// TIA Portal project "PLC Reload" (V17)

(* hardware
DEVICE "S7-1200 station_1"  S7-1200 Station
   slot 0: "Rack_0"  S7-1200 Rack  Rack  V1.0
   slot 1: "PLC_1"  CPU 1215C DC/DC/Rly  6ES7 215-1HG40-0XB0  V4.2
   slot 2: "DI 16x24VDC/DQ 16xRelay_1"  SM 1223 DI16/DQ16 x relay  6ES7 223-1PL32-0XB0  V2.0
   slot 3: "AI 4x13BIT_1"  6ES7 231-4HD32-0XB0  V2.1
*)

// ===== PLC "PLC_1"  CPU 1215C DC/DC/Rly =====

VAR_GLOBAL   // PLC tag table "Default tag table"
   "bt.Auto" AT %I0.1 : Bool;
   "CTHT_Thuan" AT %I1.2 : Bool;
   "bt.Manual" AT %I0.2 : Bool;
   "Sensor 1 Nhiệt Độ" AT %IW64 : Int;
   "Sensor 1 Độ Ảm" AT %IW66 : Int;
   "Tag_15" AT %IW11 : Int;
   "Sensor 2 Nhiệt Độ" AT %IW112 : Int;
   "Sensor 2 Độ Ảm" AT %IW114 : Int;
   "Sensor 3 Nhiệt Độ" AT %IW116 : Int;
   "Sensor 3 Độ Ảm" AT %IW118 : Int;
   "bt.BangTai" AT %I0.3 : Bool;
   "bt.Manual Đèn 1 3" AT %I0.5 : Bool;
   "bt. Cylanh Thức Ăn" AT %I0.4 : Bool;
   "CTHT_Nguoc" AT %I1.1 : Bool;
   "bt.Manual Đèn 2 4" AT %I0.6 : Bool;
   "bt.Quat" AT %I0.7 : Bool;
   "bt.PhunSuong" AT %I1.0 : Bool;
   "Đèn sưởi 1" AT %Q1.0 : Bool;
   "Băng tải 1" AT %Q1.1 : Bool;
   "#R Pump" AT %Q8.0 : Bool;
   "Xy Lanh An Duoi" AT %Q0.5 : Bool;
   "QuatAm2" AT %Q0.6 : Bool;
   "QuatAm1" AT %Q8.1 : Bool;
   "Van trên 2" AT %Q8.2 : Bool;
   "QuatThoi_Duoi" AT %Q9.1 : Bool;
   "QuatHutAm_Duoi" AT %Q9.2 : Bool;
   "Đèn sưởi 2" AT %Q0.7 : Bool;
   "#R Motor Fwd" AT %Q0.3 : Bool;
   "#R Motor Rev" AT %Q0.4 : Bool;
   "Light Green" AT %Q0.0 : Bool;
   "Light Yellow" AT %Q0.2 : Bool;
   "Băng tải 3" AT %Q9.3 : Bool;
   "Băng tải 4" AT %Q9.4 : Bool;
   "Băng tải 2" AT %Q9.0 : Bool;
   "Xylanh an tren" AT %Q8.6 : Bool;
   "Xylanh Nâng" AT %Q8.7 : Bool;
   "Tag_33" AT %Q2.4 : Bool;
   "Tag_35" AT %Q2.5 : Bool;
   "Van 3 - Bồn" AT %Q8.3 : Bool;
   "Van trên 4" AT %Q8.4 : Bool;
   "Van 1,5" AT %Q8.5 : Bool;
   "System_Byte" AT %MB100 : Byte;
   "FirstScan" AT %M100.0 : Bool;
   "DiagStatusUpdate" AT %M100.1 : Bool;
   "AlwaysTRUE" AT %M100.2 : Bool;
   "AlwaysFALSE" AT %M100.3 : Bool;
   "Clock_Byte" AT %MB110 : Byte;
   "Clock_10Hz" AT %M110.0 : Bool;
   "Clock_5Hz" AT %M110.1 : Bool;
   "Clock_2.5Hz" AT %M110.2 : Bool;
   "Clock_2Hz" AT %M110.3 : Bool;
   "Clock_1.25Hz" AT %M110.4 : Bool;
   "Clock_1Hz" AT %M110.5 : Bool;
   "Clock_0.625Hz" AT %M110.6 : Bool;
   "Clock_0.5Hz" AT %M110.7 : Bool;
   "R #01 Test" AT %M0.0 : Bool;
   "m0.7" AT %M0.1 : Bool;
   "Tag_2" AT %M10.0 : Bool;
   "Tag_6" AT %M10.1 : Bool;
   "Tag_5" AT %M10.2 : Bool;
   "Tag_8" AT %M10.3 : Bool;
   "Tag_12" AT %M10.4 : Bool;
   "Tag_13" AT %M10.5 : Bool;
   "Tag_14" AT %M10.6 : Bool;
   "Tag_16" AT %M10.7 : Bool;
   "Tag_18" AT %M11.0 : Bool;
   "R #02 Test" AT %M11.1 : Bool;
   "ND NORM_1" AT %MD200 : Real;
   "DATA NhietDo_1" AT %MD204 : Real;
   "DA NORM 1" AT %MD208 : Real;
   "DATA DoAm_1" AT %MD212 : Real;
   "Tag_22" AT %MD216 : Real;
   "ND NORM_2" AT %MD220 : Real;
   "DATA NhietDo_2" AT %MD224 : Real;
   "DA NORM 2" AT %MD228 : Real;
   "DATA DoAm_2" AT %MD232 : Real;
   "ND NORM_3" AT %MD440 : Real;
   "DATA NhietDo_3" AT %MD444 : Real;
   "DA NORM 3" AT %MD448 : Real;
   "DATA DoAm_3" AT %MD452 : Real;
   "Auto Mode" AT %M1.0 : Bool;
   "Manual Mode" AT %M1.1 : Bool;
   "Cylanh Nâng" AT %M2.0 : Bool;
   "Manual Băng Tải" AT %M1.2 : Bool;
   "Băng Tải 1 2 Run" AT %M2.1 : Bool;
   "Tag_4" AT %M0.7 : Bool;
   "Tag_19" AT %M0.6 : Bool;
   "Manual Cylanh Thức Ăn" AT %M1.3 : Bool;
   "Cylanh Up Thuc Ăn" AT %M2.2 : Bool;
   "Motor FWD" AT %M2.4 : Bool;
   "Motor REV" AT %M2.5 : Bool;
   "Tag_36" AT %M6.0 : Bool;
   "Tag_37" AT %M2.3 : Bool;
   "Đèn 1 3 Manual" AT %M1.4 : Bool;
   "Đèn 2 4 Manual" AT %M1.5 : Bool;
   "Manual Quạt" AT %M1.6 : Bool;
   "Manual Phun Sương" AT %M1.7 : Bool;
   "Pump Run" AT %M2.6 : Bool;
   "Van chuong 1" AT %M2.7 : Bool;
   "Van chuong 2" AT %M3.0 : Bool;
   "Van chuong 3,4" AT %M3.1 : Bool;
   "Van 4" AT %M3.2 : Bool;
   "Van lên bồn" AT %M3.3 : Bool;
   "Auto Buổi Sáng" AT %M4.0 : Bool;
   "Auto Buổi Trưa" AT %M4.1 : Bool;
   "Auto Buổi Chiều" AT %M4.2 : Bool;
   "Auto Theo Buổi" AT %M5.0 : Bool;
   "TG_Nhiet_1" AT %M5.1 : Bool;
   "Mode Theo Buổi" AT %M5.2 : Bool;
   "Mode Cảm Biến + Theo Buổi" AT %M5.3 : Bool;
   "Tag_7" AT %MD304 : Real;
   "Tag_9" AT %MD312 : Real;
   "Tag_10" AT %MD324 : Real;
   "Tag_11" AT %MD332 : Real;
   "Tag_20" AT %MD344 : Real;
   "Tag_21" AT %MD352 : Real;
   "TG_Nhiet_2" AT %M5.4 : Bool;
   "TG_Nhiet_3" AT %M5.5 : Bool;
   "Mode Cảm Biến + Theo Buổi R" AT %M5.6 : Bool;
   "Tag_1" AT %M88.4 : Bool;
   "Tag_23" AT %M778.6 : Bool;
   "Cho an Tren" AT %M12.0 : Bool;
   "Don Ve Sinh" AT %M12.1 : Bool;
   "TG_Am_1" AT %M7.0 : Bool;
   "Tag_25" AT %MD404 : Real;
   "Tag_26" AT %MD412 : Real;
   "Tag_27" AT %MD424 : Real;
   "Tag_28" AT %MD432 : Real;
   "TG_Am_2" AT %M7.1 : Bool;
   "TG_Am_3" AT %M7.2 : Bool;
   "Tag_24" AT %M864.4 : Bool;
   "Tag_29" AT %M54.7 : Bool;
   "Sensor Pump Done" AT %I1.3 : Bool;
   "TG_Am_Quat_1" AT %M7.5 : Bool;
   "TG_Am_Quat_3" AT %M7.6 : Bool;
   "TG_Am_Quat_2" AT %M7.7 : Bool;
   "Tag_17" AT %M8.1 : Bool;
   "DonVSTren" AT %M12.2 : Bool;
END_VAR

DATA_BLOCK "Time"   // DB6
{ S7_Optimized_Access := 'TRUE' }
VERSION : 0.1
   VAR
      Reatime : DTL;
      "Dọn Vệ Sinh Trên 1" : Bool;
      Retval : Int;
      "Ăn Dưới 1" : Bool;
      "An 2" : Bool;
      "An 3" : Bool;
      "Ăn Trên 1" : Bool;
      "An Tren 2" : Bool;
      "An Tren 3" : Bool;
      "An Tren 4" : Bool;
      "An Tren 5" : Bool;
      "Dọn Vệ Sinh Dưới 1" : Bool;
      "Don VS Duoi 2" : Bool;
   END_VAR
BEGIN
END_DATA_BLOCK

DATA_BLOCK "Temp"   // DB13
{ S7_Optimized_Access := 'FALSE' }
VERSION : 0.1
   VAR
      DataNhiet1 : Real;
      DataNhiet2 : Real;
      DataNhiet3 : Real;
      DataAm1 : Real;
      DataAm2 : Real;
      DataAm3 : Real;
      SetNhiet1 : Real;
      SetNhiet2 : Real;
      SetNhiet3 : Real;
      SetAm1 : Real;
      SetAm2 : Real;
      SetAm3 : Real;
   END_VAR
BEGIN
END_DATA_BLOCK

// folder: System blocks/Program resources

DATA_BLOCK "Delay Thưc Ăn"   // DB1
{ S7_Optimized_Access := 'TRUE' }
AUTHOR : Simatic
FAMILY : IEC
NAME : IEC_TMR
VERSION : 1.0
// stored: InstanceOfName IEC_TIMER
"IEC_TIMER"
BEGIN
END_DATA_BLOCK

DATA_BLOCK "Cylanh Nâng DL"   // DB2
{ S7_Optimized_Access := 'TRUE' }
AUTHOR : Simatic
FAMILY : IEC
NAME : IEC_TMR
VERSION : 1.0
// stored: InstanceOfName IEC_TIMER
"IEC_TIMER"
BEGIN
END_DATA_BLOCK

DATA_BLOCK "Motor Check FWD"   // DB3
{ S7_Optimized_Access := 'TRUE' }
AUTHOR : Simatic
FAMILY : IEC
NAME : IEC_TMR
VERSION : 1.0
// stored: InstanceOfName IEC_TIMER
"IEC_TIMER"
BEGIN
END_DATA_BLOCK

DATA_BLOCK "Motor Check REV"   // DB4
{ S7_Optimized_Access := 'TRUE' }
AUTHOR : Simatic
FAMILY : IEC
NAME : IEC_TMR
VERSION : 1.0
// stored: InstanceOfName IEC_TIMER
"IEC_TIMER"
BEGIN
END_DATA_BLOCK

DATA_BLOCK "Delay Pump"   // DB5
{ S7_Optimized_Access := 'TRUE' }
AUTHOR : Simatic
FAMILY : IEC
NAME : IEC_TMR
VERSION : 1.0
// stored: InstanceOfName IEC_TIMER
"IEC_TIMER"
BEGIN
END_DATA_BLOCK

DATA_BLOCK "Dl Time"   // DB7
{ S7_Optimized_Access := 'TRUE' }
AUTHOR : Simatic
FAMILY : IEC
NAME : IEC_TMR
VERSION : 1.0
// stored: InstanceOfName IEC_TIMER
"IEC_TIMER"
BEGIN
END_DATA_BLOCK

DATA_BLOCK "Dl Don Ve Sinh"   // DB8
{ S7_Optimized_Access := 'TRUE' }
AUTHOR : Simatic
FAMILY : IEC
NAME : IEC_TMR
VERSION : 1.0
// stored: InstanceOfName IEC_TIMER
"IEC_TIMER"
BEGIN
END_DATA_BLOCK

DATA_BLOCK "Dl Off"   // DB9
{ S7_Optimized_Access := 'TRUE' }
AUTHOR : Simatic
FAMILY : IEC
NAME : IEC_TMR
VERSION : 1.0
// stored: InstanceOfName IEC_TIMER
"IEC_TIMER"
BEGIN
END_DATA_BLOCK

DATA_BLOCK "DL Off 2"   // DB10
{ S7_Optimized_Access := 'TRUE' }
AUTHOR : Simatic
FAMILY : IEC
NAME : IEC_TMR
VERSION : 1.0
// stored: InstanceOfName IEC_TIMER
"IEC_TIMER"
BEGIN
END_DATA_BLOCK

DATA_BLOCK "DLOff 3"   // DB11
{ S7_Optimized_Access := 'TRUE' }
AUTHOR : Simatic
FAMILY : IEC
NAME : IEC_TMR
VERSION : 1.0
// stored: InstanceOfName IEC_TIMER
"IEC_TIMER"
BEGIN
END_DATA_BLOCK

DATA_BLOCK "DL Off Time An"   // DB12
{ S7_Optimized_Access := 'TRUE' }
AUTHOR : Simatic
FAMILY : IEC
NAME : IEC_TMR
VERSION : 1.0
// stored: InstanceOfName IEC_TIMER
"IEC_TIMER"
BEGIN
END_DATA_BLOCK

DATA_BLOCK "VESINH"   // DB14
{ S7_Optimized_Access := 'TRUE' }
AUTHOR : Simatic
FAMILY : IEC
NAME : IEC_TMR
VERSION : 1.0
// stored: InstanceOfName IEC_TIMER
"IEC_TIMER"
BEGIN
END_DATA_BLOCK

// folder: (top level)

FUNCTION "MC_Output" : Void   // FC1, LAD
{ S7_Optimized_Access := 'TRUE' }
VERSION : 0.1
BEGIN

REGION Network 1
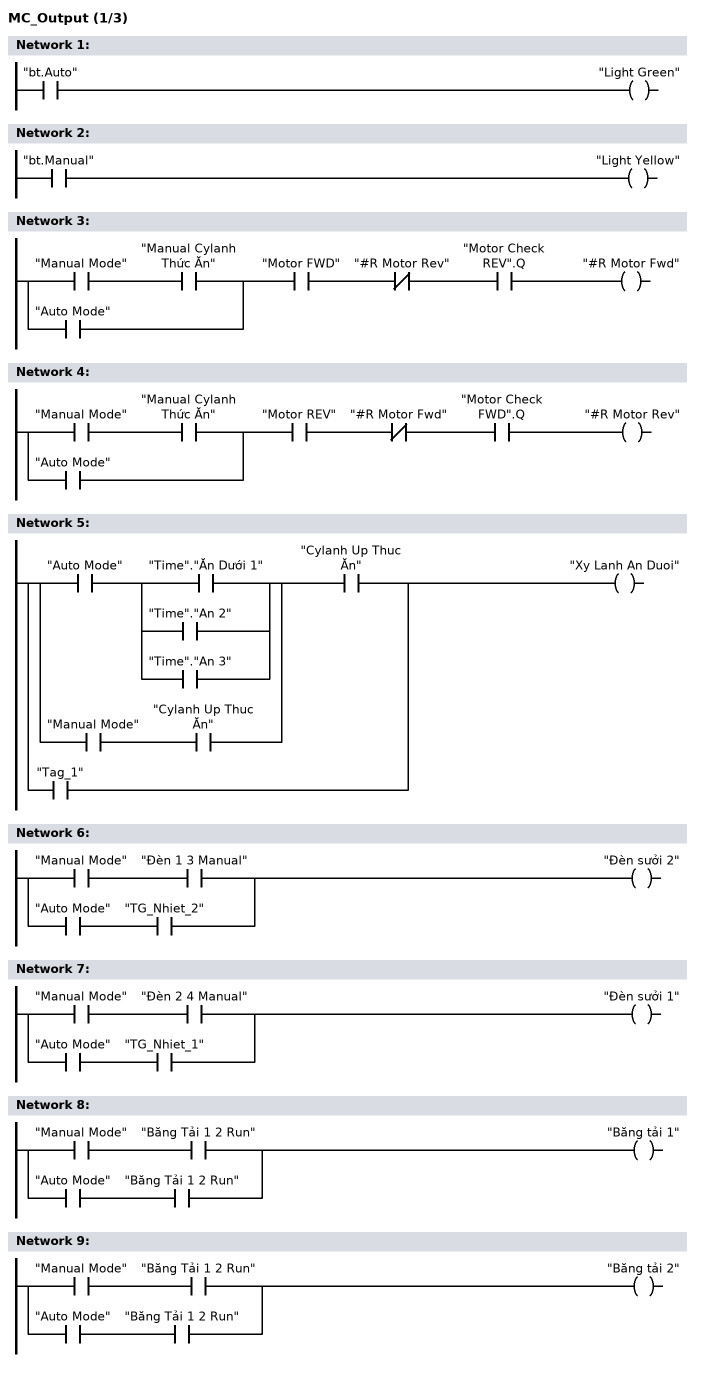
   RUNG wire#powerrail
      Contact( "bt.Auto" )
      Coil( "Light Green" )
   END_RUNG
   // the same network as SCL:
   "Light Green" := "bt.Auto";
END_REGION

REGION Network 2
   RUNG wire#powerrail
      Contact( "bt.Manual" )
      Coil( "Light Yellow" )
   END_RUNG
   // the same network as SCL:
   "Light Yellow" := "bt.Manual";
END_REGION

REGION Network 3
   RUNG wire#powerrail
      Contact( "Manual Mode" )
      Contact( "Manual Cylanh Thức Ăn" )
      wire#w1
      Contact( "Motor FWD" )
      I_Contact( "#R Motor Rev" )
      Contact( "Motor Check REV".Q )
      Coil( "#R Motor Fwd" )
   END_RUNG
   RUNG wire#powerrail
      Contact( "Auto Mode" )
   END_RUNG wire#w1
   // the same network as SCL:
   "#R Motor Fwd" := (("Manual Mode" AND "Manual Cylanh Thức Ăn") OR "Auto Mode") AND "Motor FWD" AND NOT "#R Motor Rev" AND "Motor Check REV".Q;
END_REGION

REGION Network 4
   RUNG wire#powerrail
      Contact( "Manual Mode" )
      Contact( "Manual Cylanh Thức Ăn" )
      wire#w1
      Contact( "Motor REV" )
      I_Contact( "#R Motor Fwd" )
      Contact( "Motor Check FWD".Q )
      Coil( "#R Motor Rev" )
   END_RUNG
   RUNG wire#powerrail
      Contact( "Auto Mode" )
   END_RUNG wire#w1
   // the same network as SCL:
   "#R Motor Rev" := (("Manual Mode" AND "Manual Cylanh Thức Ăn") OR "Auto Mode") AND "Motor REV" AND NOT "#R Motor Fwd" AND "Motor Check FWD".Q;
END_REGION

REGION Network 5
   RUNG wire#powerrail
      Contact( "Auto Mode" )
      wire#w1
      Contact( "Time"."Ăn Dưới 1" )
      wire#w2
      Contact( "Cylanh Up Thuc Ăn" )
      wire#w3
      Coil( "Xy Lanh An Duoi" )
   END_RUNG
   RUNG wire#w1
      Contact( "Time"."An 2" )
   END_RUNG wire#w2
   RUNG wire#w1
      Contact( "Time"."An 3" )
   END_RUNG wire#w2
   RUNG wire#powerrail
      Contact( "Manual Mode" )
      Contact( "Cylanh Up Thuc Ăn" )
   END_RUNG wire#w2
   RUNG wire#powerrail
      Contact( "Tag_1" )
   END_RUNG wire#w3
   // the same network as SCL:
   "Xy Lanh An Duoi" := ((("Auto Mode" AND ("Time"."Ăn Dưới 1" OR "Time"."An 2" OR "Time"."An 3")) OR ("Manual Mode" AND "Cylanh Up Thuc Ăn")) AND "Cylanh Up Thuc Ăn") OR "Tag_1";
END_REGION

REGION Network 6
   RUNG wire#powerrail
      Contact( "Manual Mode" )
      Contact( "Đèn 1 3 Manual" )
      wire#w1
      Coil( "Đèn sưởi 2" )
   END_RUNG
   RUNG wire#powerrail
      Contact( "Auto Mode" )
      Contact( "TG_Nhiet_2" )
   END_RUNG wire#w1
   // the same network as SCL:
   "Đèn sưởi 2" := ("Manual Mode" AND "Đèn 1 3 Manual") OR ("Auto Mode" AND "TG_Nhiet_2");
END_REGION

REGION Network 7
   RUNG wire#powerrail
      Contact( "Manual Mode" )
      Contact( "Đèn 2 4 Manual" )
      wire#w1
      Coil( "Đèn sưởi 1" )
   END_RUNG
   RUNG wire#powerrail
      Contact( "Auto Mode" )
      Contact( "TG_Nhiet_1" )
   END_RUNG wire#w1
   // the same network as SCL:
   "Đèn sưởi 1" := ("Manual Mode" AND "Đèn 2 4 Manual") OR ("Auto Mode" AND "TG_Nhiet_1");
END_REGION

REGION Network 8
   RUNG wire#powerrail
      Contact( "Manual Mode" )
      Contact( "Băng Tải 1 2 Run" )
      wire#w1
      Coil( "Băng tải 1" )
   END_RUNG
   RUNG wire#powerrail
      Contact( "Auto Mode" )
      Contact( "Băng Tải 1 2 Run" )
   END_RUNG wire#w1
   // the same network as SCL:
   "Băng tải 1" := ("Manual Mode" AND "Băng Tải 1 2 Run") OR ("Auto Mode" AND "Băng Tải 1 2 Run");
END_REGION

REGION Network 9
   RUNG wire#powerrail
      Contact( "Manual Mode" )
      Contact( "Băng Tải 1 2 Run" )
      wire#w1
      Coil( "Băng tải 2" )
   END_RUNG
   RUNG wire#powerrail
      Contact( "Auto Mode" )
      Contact( "Băng Tải 1 2 Run" )
   END_RUNG wire#w1
   // the same network as SCL:
   "Băng tải 2" := ("Manual Mode" AND "Băng Tải 1 2 Run") OR ("Auto Mode" AND "Băng Tải 1 2 Run");
END_REGION

REGION Network 10
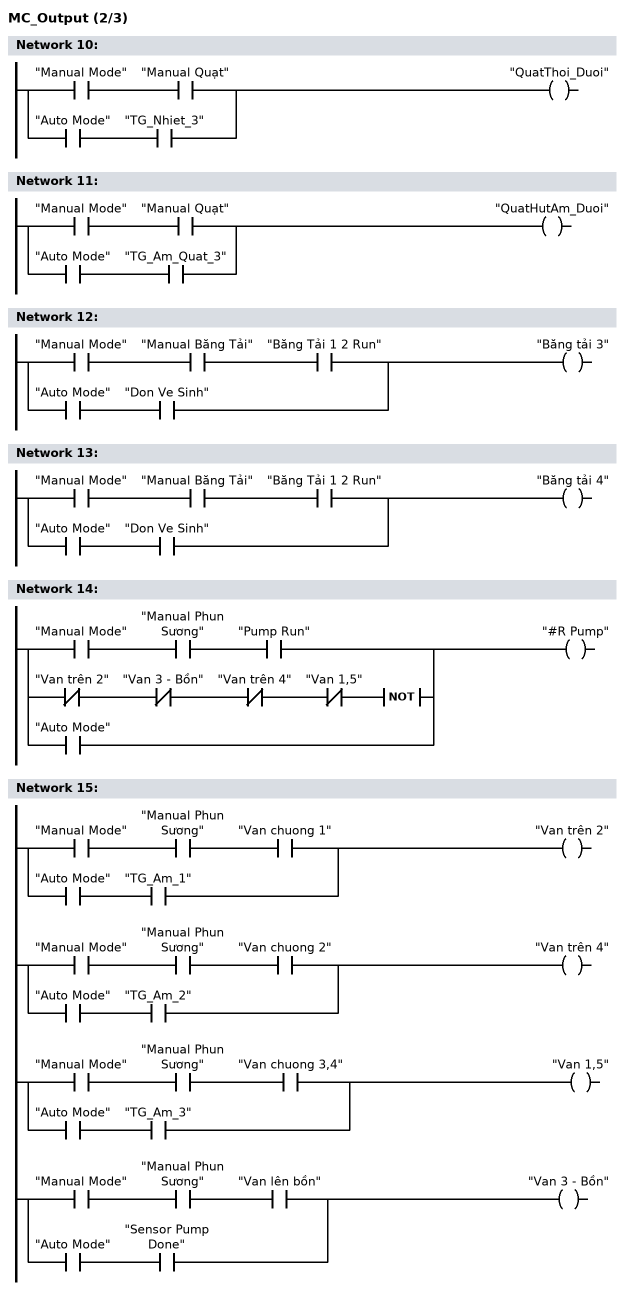
   RUNG wire#powerrail
      Contact( "Manual Mode" )
      Contact( "Manual Quạt" )
      wire#w1
      Coil( "QuatThoi_Duoi" )
   END_RUNG
   RUNG wire#powerrail
      Contact( "Auto Mode" )
      Contact( "TG_Nhiet_3" )
   END_RUNG wire#w1
   // the same network as SCL:
   "QuatThoi_Duoi" := ("Manual Mode" AND "Manual Quạt") OR ("Auto Mode" AND "TG_Nhiet_3");
END_REGION

REGION Network 11
   RUNG wire#powerrail
      Contact( "Manual Mode" )
      Contact( "Manual Quạt" )
      wire#w1
      Coil( "QuatHutAm_Duoi" )
   END_RUNG
   RUNG wire#powerrail
      Contact( "Auto Mode" )
      Contact( "TG_Am_Quat_3" )
   END_RUNG wire#w1
   // the same network as SCL:
   "QuatHutAm_Duoi" := ("Manual Mode" AND "Manual Quạt") OR ("Auto Mode" AND "TG_Am_Quat_3");
END_REGION

REGION Network 12
   RUNG wire#powerrail
      Contact( "Manual Mode" )
      Contact( "Manual Băng Tải" )
      Contact( "Băng Tải 1 2 Run" )
      wire#w1
      Coil( "Băng tải 3" )
   END_RUNG
   RUNG wire#powerrail
      Contact( "Auto Mode" )
      Contact( "Don Ve Sinh" )
   END_RUNG wire#w1
   // the same network as SCL:
   "Băng tải 3" := ("Manual Mode" AND "Manual Băng Tải" AND "Băng Tải 1 2 Run") OR ("Auto Mode" AND "Don Ve Sinh");
END_REGION

REGION Network 13
   RUNG wire#powerrail
      Contact( "Manual Mode" )
      Contact( "Manual Băng Tải" )
      Contact( "Băng Tải 1 2 Run" )
      wire#w1
      Coil( "Băng tải 4" )
   END_RUNG
   RUNG wire#powerrail
      Contact( "Auto Mode" )
      Contact( "Don Ve Sinh" )
   END_RUNG wire#w1
   // the same network as SCL:
   "Băng tải 4" := ("Manual Mode" AND "Manual Băng Tải" AND "Băng Tải 1 2 Run") OR ("Auto Mode" AND "Don Ve Sinh");
END_REGION

REGION Network 14
   RUNG wire#powerrail
      Contact( "Manual Mode" )
      Contact( "Manual Phun Sương" )
      Contact( "Pump Run" )
      wire#w1
      Coil( "#R Pump" )
   END_RUNG
   RUNG wire#powerrail
      I_Contact( "Van trên 2" )
      I_Contact( "Van 3 - Bồn" )
      I_Contact( "Van trên 4" )
      I_Contact( "Van 1,5" )
      Not()
   END_RUNG wire#w1
   RUNG wire#powerrail
      Contact( "Auto Mode" )
   END_RUNG wire#w1
   // the same network as SCL:
   "#R Pump" := ("Manual Mode" AND "Manual Phun Sương" AND "Pump Run") OR NOT (NOT "Van trên 2" AND NOT "Van 3 - Bồn" AND NOT "Van trên 4" AND NOT "Van 1,5") OR "Auto Mode";
END_REGION

REGION Network 15
   RUNG wire#powerrail
      Contact( "Manual Mode" )
      Contact( "Manual Phun Sương" )
      Contact( "Van chuong 1" )
      wire#w1
      Coil( "Van trên 2" )
   END_RUNG
   RUNG wire#powerrail
      Contact( "Auto Mode" )
      Contact( "TG_Am_1" )
   END_RUNG wire#w1
   RUNG wire#powerrail
      Contact( "Manual Mode" )
      Contact( "Manual Phun Sương" )
      Contact( "Van chuong 2" )
      wire#w2
      Coil( "Van trên 4" )
   END_RUNG
   RUNG wire#powerrail
      Contact( "Auto Mode" )
      Contact( "TG_Am_2" )
   END_RUNG wire#w2
   RUNG wire#powerrail
      Contact( "Manual Mode" )
      Contact( "Manual Phun Sương" )
      Contact( "Van chuong 3,4" )
      wire#w3
      Coil( "Van 1,5" )
   END_RUNG
   RUNG wire#powerrail
      Contact( "Auto Mode" )
      Contact( "TG_Am_3" )
   END_RUNG wire#w3
   RUNG wire#powerrail
      Contact( "Manual Mode" )
      Contact( "Manual Phun Sương" )
      Contact( "Van lên bồn" )
      wire#w4
      Coil( "Van 3 - Bồn" )
   END_RUNG
   RUNG wire#powerrail
      Contact( "Auto Mode" )
      Contact( "Sensor Pump Done" )
   END_RUNG wire#w4
   // the same network as SCL:
   "Van trên 2" := ("Manual Mode" AND "Manual Phun Sương" AND "Van chuong 1") OR ("Auto Mode" AND "TG_Am_1");
   "Van trên 4" := ("Manual Mode" AND "Manual Phun Sương" AND "Van chuong 2") OR ("Auto Mode" AND "TG_Am_2");
   "Van 1,5" := ("Manual Mode" AND "Manual Phun Sương" AND "Van chuong 3,4") OR ("Auto Mode" AND "TG_Am_3");
   "Van 3 - Bồn" := ("Manual Mode" AND "Manual Phun Sương" AND "Van lên bồn") OR ("Auto Mode" AND "Sensor Pump Done");
END_REGION

REGION Network 17
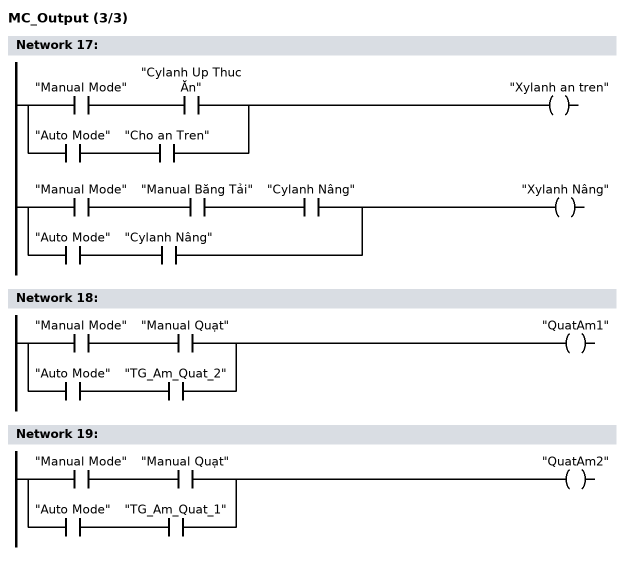
   RUNG wire#powerrail
      Contact( "Manual Mode" )
      Contact( "Cylanh Up Thuc Ăn" )
      wire#w1
      Coil( "Xylanh an tren" )
   END_RUNG
   RUNG wire#powerrail
      Contact( "Auto Mode" )
      Contact( "Cho an Tren" )
   END_RUNG wire#w1
   RUNG wire#powerrail
      Contact( "Manual Mode" )
      Contact( "Manual Băng Tải" )
      Contact( "Cylanh Nâng" )
      wire#w2
      Coil( "Xylanh Nâng" )
   END_RUNG
   RUNG wire#powerrail
      Contact( "Auto Mode" )
      Contact( "Cylanh Nâng" )
   END_RUNG wire#w2
   // the same network as SCL:
   "Xylanh an tren" := ("Manual Mode" AND "Cylanh Up Thuc Ăn") OR ("Auto Mode" AND "Cho an Tren");
   "Xylanh Nâng" := ("Manual Mode" AND "Manual Băng Tải" AND "Cylanh Nâng") OR ("Auto Mode" AND "Cylanh Nâng");
END_REGION

REGION Network 18
   RUNG wire#powerrail
      Contact( "Manual Mode" )
      Contact( "Manual Quạt" )
      wire#w1
      Coil( "QuatAm1" )
   END_RUNG
   RUNG wire#powerrail
      Contact( "Auto Mode" )
      Contact( "TG_Am_Quat_2" )
   END_RUNG wire#w1
   // the same network as SCL:
   "QuatAm1" := ("Manual Mode" AND "Manual Quạt") OR ("Auto Mode" AND "TG_Am_Quat_2");
END_REGION

REGION Network 19
   RUNG wire#powerrail
      Contact( "Manual Mode" )
      Contact( "Manual Quạt" )
      wire#w1
      Coil( "QuatAm2" )
   END_RUNG
   RUNG wire#powerrail
      Contact( "Auto Mode" )
      Contact( "TG_Am_Quat_1" )
   END_RUNG wire#w1
   // the same network as SCL:
   "QuatAm2" := ("Manual Mode" AND "Manual Quạt") OR ("Auto Mode" AND "TG_Am_Quat_1");
END_REGION
END_FUNCTION

FUNCTION "MC_Input" : Void   // FC2, LAD
{ S7_Optimized_Access := 'TRUE' }
VERSION : 0.1
BEGIN

REGION Network 1
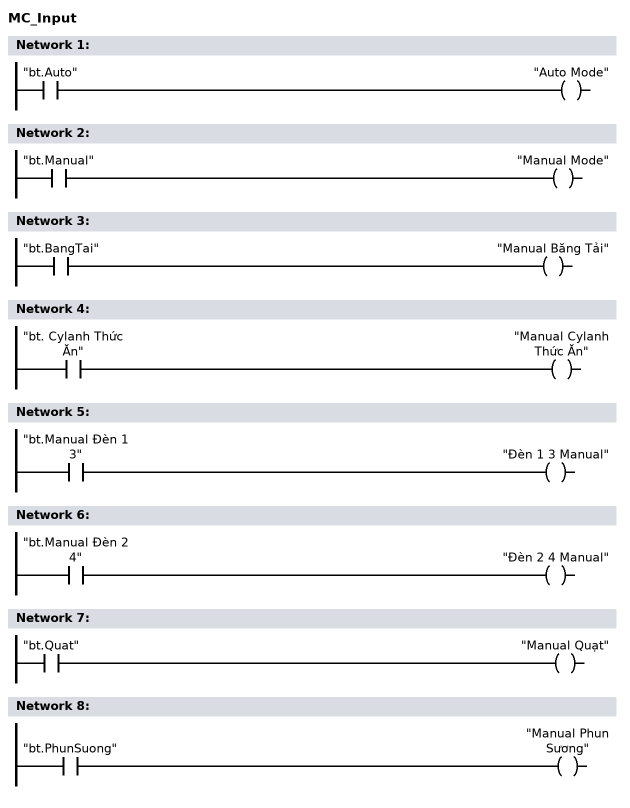
   RUNG wire#powerrail
      Contact( "bt.Auto" )
      Coil( "Auto Mode" )
   END_RUNG
   // the same network as SCL:
   "Auto Mode" := "bt.Auto";
END_REGION

REGION Network 2
   RUNG wire#powerrail
      Contact( "bt.Manual" )
      Coil( "Manual Mode" )
   END_RUNG
   // the same network as SCL:
   "Manual Mode" := "bt.Manual";
END_REGION

REGION Network 3
   RUNG wire#powerrail
      Contact( "bt.BangTai" )
      Coil( "Manual Băng Tải" )
   END_RUNG
   // the same network as SCL:
   "Manual Băng Tải" := "bt.BangTai";
END_REGION

REGION Network 4
   RUNG wire#powerrail
      Contact( "bt. Cylanh Thức Ăn" )
      Coil( "Manual Cylanh Thức Ăn" )
   END_RUNG
   // the same network as SCL:
   "Manual Cylanh Thức Ăn" := "bt. Cylanh Thức Ăn";
END_REGION

REGION Network 5
   RUNG wire#powerrail
      Contact( "bt.Manual Đèn 1 3" )
      Coil( "Đèn 1 3 Manual" )
   END_RUNG
   // the same network as SCL:
   "Đèn 1 3 Manual" := "bt.Manual Đèn 1 3";
END_REGION

REGION Network 6
   RUNG wire#powerrail
      Contact( "bt.Manual Đèn 2 4" )
      Coil( "Đèn 2 4 Manual" )
   END_RUNG
   // the same network as SCL:
   "Đèn 2 4 Manual" := "bt.Manual Đèn 2 4";
END_REGION

REGION Network 7
   RUNG wire#powerrail
      Contact( "bt.Quat" )
      Coil( "Manual Quạt" )
   END_RUNG
   // the same network as SCL:
   "Manual Quạt" := "bt.Quat";
END_REGION

REGION Network 8
   RUNG wire#powerrail
      Contact( "bt.PhunSuong" )
      Coil( "Manual Phun Sương" )
   END_RUNG
   // the same network as SCL:
   "Manual Phun Sương" := "bt.PhunSuong";
END_REGION
END_FUNCTION

FUNCTION "MC_Read Sensor 1" : Void   // FC3, LAD
{ S7_Optimized_Access := 'TRUE' }
VERSION : 0.1
BEGIN

REGION Network 1
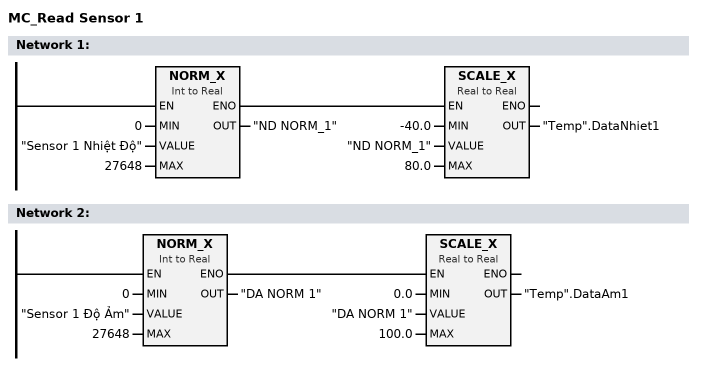
   RUNG wire#powerrail
      { S7_Templates := "[SrcType := Int, DestType := Real]" } Normalize(min := 0, value := "Sensor 1 Nhiệt Độ", max := 27648, out => "ND NORM_1")
      { S7_Templates := "[SrcType := Real, DestType := Real]" } Scale(min := -40.0, value := "ND NORM_1", max := 80.0, out => "Temp".DataNhiet1)
   END_RUNG
   // the same network as SCL:
   "ND NORM_1" := NORM_X(MIN := 0, VALUE := "Sensor 1 Nhiệt Độ", MAX := 27648);
   "Temp".DataNhiet1 := SCALE_X(MIN := -40.0, VALUE := "ND NORM_1", MAX := 80.0);
END_REGION

REGION Network 2
   RUNG wire#powerrail
      { S7_Templates := "[SrcType := Int, DestType := Real]" } Normalize(min := 0, value := "Sensor 1 Độ Ảm", max := 27648, out => "DA NORM 1")
      { S7_Templates := "[SrcType := Real, DestType := Real]" } Scale(min := 0.0, value := "DA NORM 1", max := 100.0, out => "Temp".DataAm1)
   END_RUNG
   // the same network as SCL:
   "DA NORM 1" := NORM_X(MIN := 0, VALUE := "Sensor 1 Độ Ảm", MAX := 27648);
   "Temp".DataAm1 := SCALE_X(MIN := 0.0, VALUE := "DA NORM 1", MAX := 100.0);
END_REGION
END_FUNCTION

FUNCTION "MC_Read Sensor 2" : Void   // FC4, LAD
{ S7_Optimized_Access := 'TRUE' }
VERSION : 0.1
BEGIN

REGION Network 1
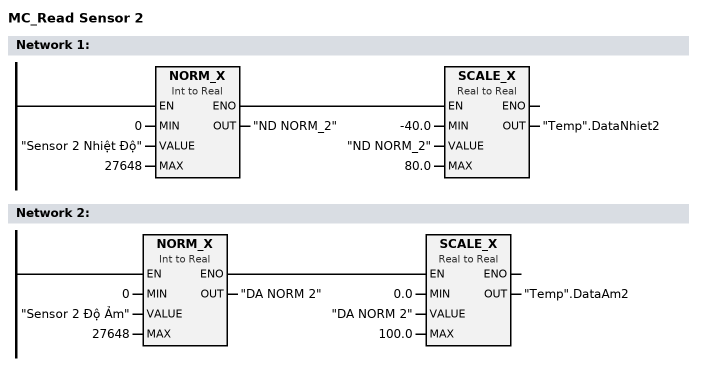
   RUNG wire#powerrail
      { S7_Templates := "[SrcType := Int, DestType := Real]" } Normalize(min := 0, value := "Sensor 2 Nhiệt Độ", max := 27648, out => "ND NORM_2")
      { S7_Templates := "[SrcType := Real, DestType := Real]" } Scale(min := -40.0, value := "ND NORM_2", max := 80.0, out => "Temp".DataNhiet2)
   END_RUNG
   // the same network as SCL:
   "ND NORM_2" := NORM_X(MIN := 0, VALUE := "Sensor 2 Nhiệt Độ", MAX := 27648);
   "Temp".DataNhiet2 := SCALE_X(MIN := -40.0, VALUE := "ND NORM_2", MAX := 80.0);
END_REGION

REGION Network 2
   RUNG wire#powerrail
      { S7_Templates := "[SrcType := Int, DestType := Real]" } Normalize(min := 0, value := "Sensor 2 Độ Ảm", max := 27648, out => "DA NORM 2")
      { S7_Templates := "[SrcType := Real, DestType := Real]" } Scale(min := 0.0, value := "DA NORM 2", max := 100.0, out => "Temp".DataAm2)
   END_RUNG
   // the same network as SCL:
   "DA NORM 2" := NORM_X(MIN := 0, VALUE := "Sensor 2 Độ Ảm", MAX := 27648);
   "Temp".DataAm2 := SCALE_X(MIN := 0.0, VALUE := "DA NORM 2", MAX := 100.0);
END_REGION
END_FUNCTION

FUNCTION "MC_Read Sensor 3" : Void   // FC5, LAD
{ S7_Optimized_Access := 'TRUE' }
VERSION : 0.1
BEGIN

REGION Network 1
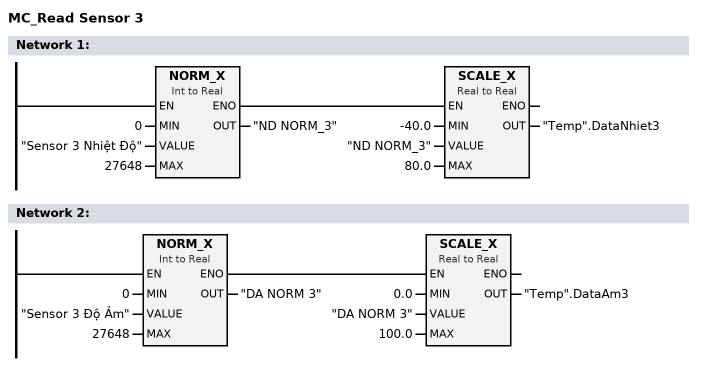
   RUNG wire#powerrail
      { S7_Templates := "[SrcType := Int, DestType := Real]" } Normalize(min := 0, value := "Sensor 3 Nhiệt Độ", max := 27648, out => "ND NORM_3")
      { S7_Templates := "[SrcType := Real, DestType := Real]" } Scale(min := -40.0, value := "ND NORM_3", max := 80.0, out => "Temp".DataNhiet3)
   END_RUNG
   // the same network as SCL:
   "ND NORM_3" := NORM_X(MIN := 0, VALUE := "Sensor 3 Nhiệt Độ", MAX := 27648);
   "Temp".DataNhiet3 := SCALE_X(MIN := -40.0, VALUE := "ND NORM_3", MAX := 80.0);
END_REGION

REGION Network 2
   RUNG wire#powerrail
      { S7_Templates := "[SrcType := Int, DestType := Real]" } Normalize(min := 0, value := "Sensor 3 Độ Ảm", max := 27648, out => "DA NORM 3")
      { S7_Templates := "[SrcType := Real, DestType := Real]" } Scale(min := 0.0, value := "DA NORM 3", max := 100.0, out => "Temp".DataAm3)
   END_RUNG
   // the same network as SCL:
   "DA NORM 3" := NORM_X(MIN := 0, VALUE := "Sensor 3 Độ Ảm", MAX := 27648);
   "Temp".DataAm3 := SCALE_X(MIN := 0.0, VALUE := "DA NORM 3", MAX := 100.0);
END_REGION
END_FUNCTION

FUNCTION "MC_Control" : Void   // FC7, LAD
{ S7_Optimized_Access := 'TRUE' }
VERSION : 0.1
   VAR_TEMP   // added for the SCL form of the ladder/FBD networks
      _w1 : Bool;
   END_VAR
BEGIN

REGION Network 1
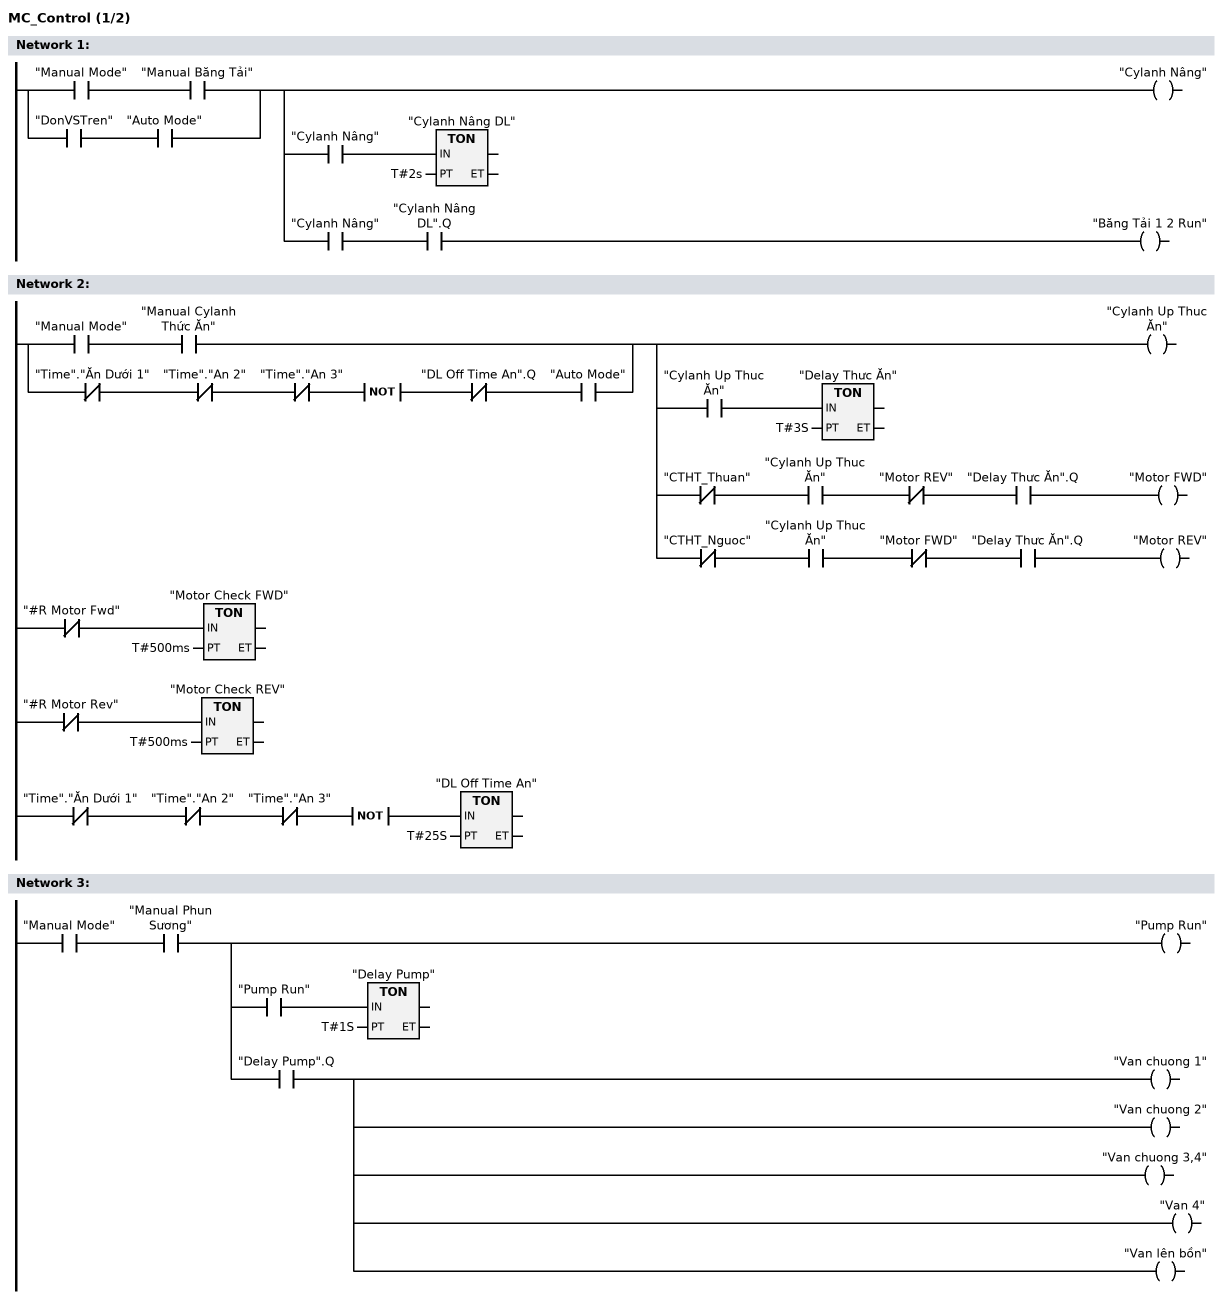
   "Cylanh Nâng" := ("Manual Mode" AND "Manual Băng Tải") OR ("DonVSTren" AND "Auto Mode");
   "Cylanh Nâng DL".TON(IN := "Cylanh Nâng" AND "Cylanh Nâng", PT := T#2s);
   "Băng Tải 1 2 Run" := "Cylanh Nâng" AND "Cylanh Nâng" AND "Cylanh Nâng DL".Q;
END_REGION

REGION Network 2
   "Cylanh Up Thuc Ăn" := ("Manual Mode" AND "Manual Cylanh Thức Ăn") OR (NOT (NOT "Time"."Ăn Dưới 1" AND NOT "Time"."An 2" AND NOT "Time"."An 3") AND NOT "DL Off Time An".Q AND "Auto Mode");
   "Delay Thưc Ăn".TON(IN := "Cylanh Up Thuc Ăn" AND "Cylanh Up Thuc Ăn", PT := T#3S);
   "Motor FWD" := "Cylanh Up Thuc Ăn" AND NOT "CTHT_Thuan" AND "Cylanh Up Thuc Ăn" AND NOT "Motor REV" AND "Delay Thưc Ăn".Q;
   "Motor REV" := "Cylanh Up Thuc Ăn" AND NOT "CTHT_Nguoc" AND "Cylanh Up Thuc Ăn" AND NOT "Motor FWD" AND "Delay Thưc Ăn".Q;
   "Motor Check FWD".TON(IN := NOT "#R Motor Fwd", PT := T#500ms);
   "Motor Check REV".TON(IN := NOT "#R Motor Rev", PT := T#500ms);
   "DL Off Time An".TON(IN := NOT (NOT "Time"."Ăn Dưới 1" AND NOT "Time"."An 2" AND NOT "Time"."An 3"),
                        PT := T#25S);
END_REGION

REGION Network 3
   "Pump Run" := "Manual Mode" AND "Manual Phun Sương";
   "Delay Pump".TON(IN := "Pump Run" AND "Pump Run", PT := T#1S);
   "Van chuong 1" := "Pump Run" AND "Delay Pump".Q;
   "Van chuong 2" := "Van chuong 1";
   "Van chuong 3,4" := "Van chuong 1";
   "Van 4" := "Van chuong 1";
   "Van lên bồn" := "Van chuong 1";
END_REGION

REGION Network 4
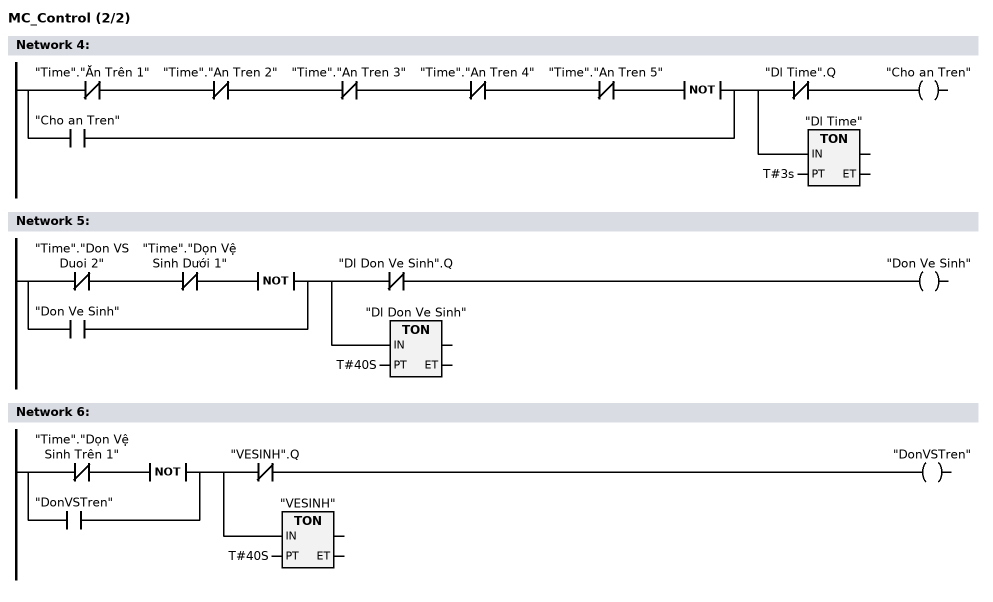
   #_w1 := NOT (NOT "Time"."Ăn Trên 1" AND NOT "Time"."An Tren 2" AND NOT "Time"."An Tren 3" AND NOT "Time"."An Tren 4" AND NOT "Time"."An Tren 5") OR "Cho an Tren";
   "Cho an Tren" := #_w1 AND NOT "Dl Time".Q;
   "Dl Time".TON(IN := #_w1, PT := T#3s);
END_REGION

REGION Network 5
   #_w1 := NOT (NOT "Time"."Don VS Duoi 2" AND NOT "Time"."Dọn Vệ Sinh Dưới 1") OR "Don Ve Sinh";
   "Don Ve Sinh" := #_w1 AND NOT "Dl Don Ve Sinh".Q;
   "Dl Don Ve Sinh".TON(IN := #_w1, PT := T#40S);
END_REGION

REGION Network 6
   #_w1 := NOT (NOT "Time"."Dọn Vệ Sinh Trên 1") OR "DonVSTren";
   "DonVSTren" := #_w1 AND NOT "VESINH".Q;
   "VESINH".TON(IN := #_w1, PT := T#40S);
END_REGION
END_FUNCTION

FUNCTION "MC_Auto" : Void   // FC8, LAD
{ S7_Optimized_Access := 'TRUE' }
VERSION : 0.1
   VAR_TEMP   // added for the SCL form of the ladder/FBD networks
      _w1 : Bool;
      _w2 : Bool;
      _w3 : Bool;
   END_VAR
BEGIN

REGION Network 1
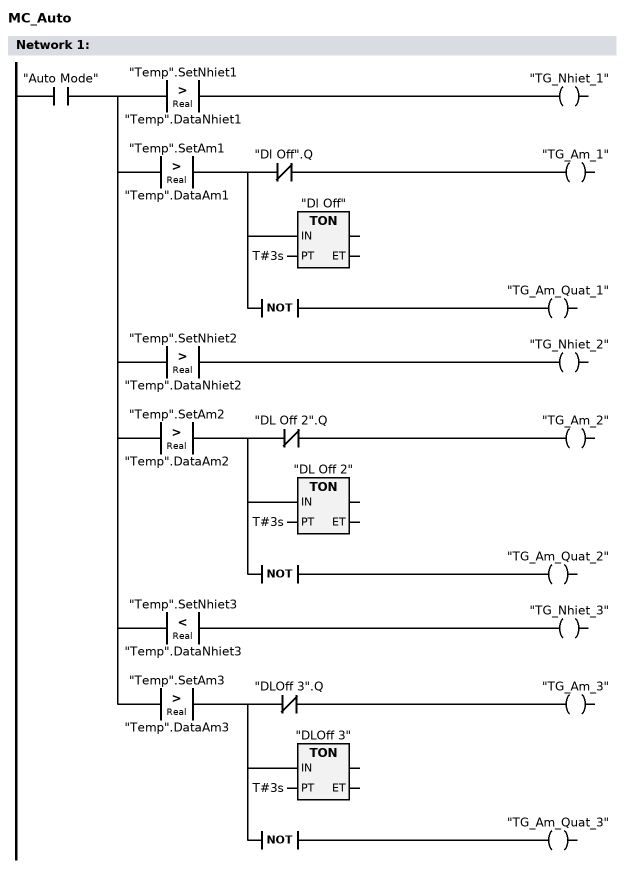
   "TG_Nhiet_1" := "Auto Mode" AND ("Temp".SetNhiet1 > "Temp".DataNhiet1);
   #_w1 := "Auto Mode" AND ("Temp".SetAm1 > "Temp".DataAm1);
   "TG_Am_1" := #_w1 AND NOT "Dl Off".Q;
   "Dl Off".TON(IN := #_w1, PT := T#3s);
   "TG_Am_Quat_1" := NOT #_w1;
   "TG_Nhiet_2" := "Auto Mode" AND ("Temp".SetNhiet2 > "Temp".DataNhiet2);
   #_w2 := "Auto Mode" AND ("Temp".SetAm2 > "Temp".DataAm2);
   "TG_Am_2" := #_w2 AND NOT "DL Off 2".Q;
   "DL Off 2".TON(IN := #_w2, PT := T#3s);
   "TG_Am_Quat_2" := NOT #_w2;
   "TG_Nhiet_3" := "Auto Mode" AND ("Temp".SetNhiet3 < "Temp".DataNhiet3);
   #_w3 := "Auto Mode" AND ("Temp".SetAm3 > "Temp".DataAm3);
   "TG_Am_3" := #_w3 AND NOT "DLOff 3".Q;
   "DLOff 3".TON(IN := #_w3, PT := T#3s);
   "TG_Am_Quat_3" := NOT #_w3;
END_REGION
END_FUNCTION

FUNCTION "MC_Settime" : Void   // FC9, LAD
{ S7_Optimized_Access := 'TRUE' }
VERSION : 0.1
BEGIN

REGION Network 1
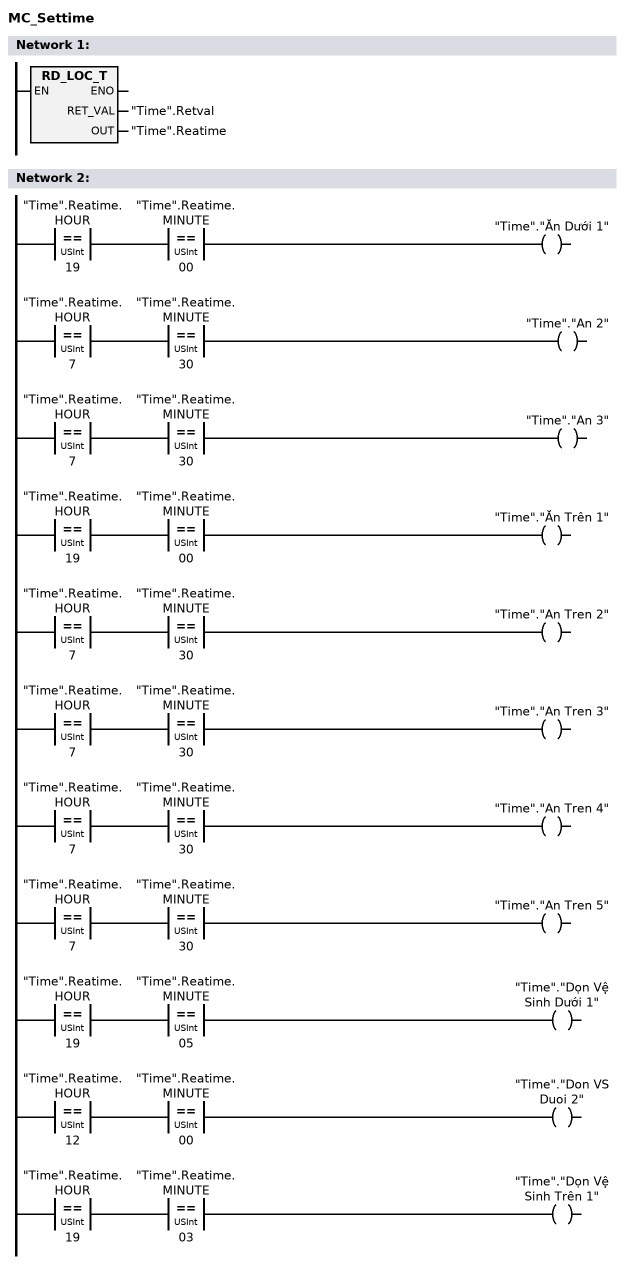
   "Time".Retval := RD_LOC_T(OUT => "Time".Reatime);
END_REGION

REGION Network 2
   RUNG wire#powerrail
      { S7_Templates := "SrcType := USInt" } EQ_Contact(in1 := "Time".Reatime.HOUR, in2 := 19)
      { S7_Templates := "SrcType := USInt" } EQ_Contact(in1 := "Time".Reatime.MINUTE, in2 := 00)
      Coil( "Time"."Ăn Dưới 1" )
   END_RUNG
   RUNG wire#powerrail
      { S7_Templates := "SrcType := USInt" } EQ_Contact(in1 := "Time".Reatime.HOUR, in2 := 7)
      { S7_Templates := "SrcType := USInt" } EQ_Contact(in1 := "Time".Reatime.MINUTE, in2 := 30)
      Coil( "Time"."An 2" )
   END_RUNG
   RUNG wire#powerrail
      { S7_Templates := "SrcType := USInt" } EQ_Contact(in1 := "Time".Reatime.HOUR, in2 := 7)
      { S7_Templates := "SrcType := USInt" } EQ_Contact(in1 := "Time".Reatime.MINUTE, in2 := 30)
      Coil( "Time"."An 3" )
   END_RUNG
   RUNG wire#powerrail
      { S7_Templates := "SrcType := USInt" } EQ_Contact(in1 := "Time".Reatime.HOUR, in2 := 19)
      { S7_Templates := "SrcType := USInt" } EQ_Contact(in1 := "Time".Reatime.MINUTE, in2 := 00)
      Coil( "Time"."Ăn Trên 1" )
   END_RUNG
   RUNG wire#powerrail
      { S7_Templates := "SrcType := USInt" } EQ_Contact(in1 := "Time".Reatime.HOUR, in2 := 7)
      { S7_Templates := "SrcType := USInt" } EQ_Contact(in1 := "Time".Reatime.MINUTE, in2 := 30)
      Coil( "Time"."An Tren 2" )
   END_RUNG
   RUNG wire#powerrail
      { S7_Templates := "SrcType := USInt" } EQ_Contact(in1 := "Time".Reatime.HOUR, in2 := 7)
      { S7_Templates := "SrcType := USInt" } EQ_Contact(in1 := "Time".Reatime.MINUTE, in2 := 30)
      Coil( "Time"."An Tren 3" )
   END_RUNG
   RUNG wire#powerrail
      { S7_Templates := "SrcType := USInt" } EQ_Contact(in1 := "Time".Reatime.HOUR, in2 := 7)
      { S7_Templates := "SrcType := USInt" } EQ_Contact(in1 := "Time".Reatime.MINUTE, in2 := 30)
      Coil( "Time"."An Tren 4" )
   END_RUNG
   RUNG wire#powerrail
      { S7_Templates := "SrcType := USInt" } EQ_Contact(in1 := "Time".Reatime.HOUR, in2 := 7)
      { S7_Templates := "SrcType := USInt" } EQ_Contact(in1 := "Time".Reatime.MINUTE, in2 := 30)
      Coil( "Time"."An Tren 5" )
   END_RUNG
   RUNG wire#powerrail
      { S7_Templates := "SrcType := USInt" } EQ_Contact(in1 := "Time".Reatime.HOUR, in2 := 19)
      { S7_Templates := "SrcType := USInt" } EQ_Contact(in1 := "Time".Reatime.MINUTE, in2 := 05)
      Coil( "Time"."Dọn Vệ Sinh Dưới 1" )
   END_RUNG
   RUNG wire#powerrail
      { S7_Templates := "SrcType := USInt" } EQ_Contact(in1 := "Time".Reatime.HOUR, in2 := 12)
      { S7_Templates := "SrcType := USInt" } EQ_Contact(in1 := "Time".Reatime.MINUTE, in2 := 00)
      Coil( "Time"."Don VS Duoi 2" )
   END_RUNG
   RUNG wire#powerrail
      { S7_Templates := "SrcType := USInt" } EQ_Contact(in1 := "Time".Reatime.HOUR, in2 := 19)
      { S7_Templates := "SrcType := USInt" } EQ_Contact(in1 := "Time".Reatime.MINUTE, in2 := 03)
      Coil( "Time"."Dọn Vệ Sinh Trên 1" )
   END_RUNG
   // the same network as SCL:
   "Time"."Ăn Dưới 1" := ("Time".Reatime.HOUR = 19) AND ("Time".Reatime.MINUTE = 00);
   "Time"."An 2" := ("Time".Reatime.HOUR = 7) AND ("Time".Reatime.MINUTE = 30);
   "Time"."An 3" := ("Time".Reatime.HOUR = 7) AND ("Time".Reatime.MINUTE = 30);
   "Time"."Ăn Trên 1" := ("Time".Reatime.HOUR = 19) AND ("Time".Reatime.MINUTE = 00);
   "Time"."An Tren 2" := ("Time".Reatime.HOUR = 7) AND ("Time".Reatime.MINUTE = 30);
   "Time"."An Tren 3" := ("Time".Reatime.HOUR = 7) AND ("Time".Reatime.MINUTE = 30);
   "Time"."An Tren 4" := ("Time".Reatime.HOUR = 7) AND ("Time".Reatime.MINUTE = 30);
   "Time"."An Tren 5" := ("Time".Reatime.HOUR = 7) AND ("Time".Reatime.MINUTE = 30);
   "Time"."Dọn Vệ Sinh Dưới 1" := ("Time".Reatime.HOUR = 19) AND ("Time".Reatime.MINUTE = 05);
   "Time"."Don VS Duoi 2" := ("Time".Reatime.HOUR = 12) AND ("Time".Reatime.MINUTE = 00);
   "Time"."Dọn Vệ Sinh Trên 1" := ("Time".Reatime.HOUR = 19) AND ("Time".Reatime.MINUTE = 03);
END_REGION
END_FUNCTION

ORGANIZATION_BLOCK "Main"   // OB1, LAD, ProgramCycle
TITLE = "Main Program Sweep (Cycle)"
{ S7_Optimized_Access := 'TRUE' }
VERSION : 0.1
   VAR_INPUT
      Initial_Call : Bool;   // Initial call of this OB
      Remanence : Bool;   // =True, if remanent data are available
   END_VAR
   VAR_TEMP
      ok : Int;
   END_VAR
   VAR_TEMP   // added for the SCL form of the ladder/FBD networks
      _w1 : Bool;
      _w2 : Bool;
      _w3 : Bool;
      _w4 : Bool;
   END_VAR
BEGIN

REGION Network 1
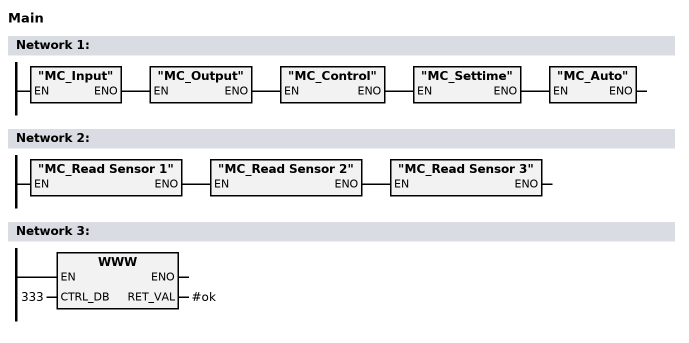
   RUNG wire#powerrail
      "MC_Input"()
      "MC_Output"()
      "MC_Control"()
      "MC_Settime"()
      "MC_Auto"()
   END_RUNG
   // the same network as SCL:
   "MC_Input"(ENO => #_w1);
   "MC_Output"(EN := #_w1, ENO => #_w2);
   "MC_Control"(EN := #_w2, ENO => #_w3);
   "MC_Settime"(EN := #_w3, ENO => #_w4);
   IF #_w4 THEN "MC_Auto"(); END_IF;
END_REGION

REGION Network 2
   RUNG wire#powerrail
      "MC_Read Sensor 1"()
      "MC_Read Sensor 2"()
      "MC_Read Sensor 3"()
   END_RUNG
   // the same network as SCL:
   "MC_Read Sensor 1"(ENO => #_w1);
   "MC_Read Sensor 2"(EN := #_w1, ENO => #_w2);
   IF #_w2 THEN "MC_Read Sensor 3"(); END_IF;
END_REGION

REGION Network 3
   #ok := WWW(CTRL_DB := 333);
END_REGION
END_ORGANIZATION_BLOCK